VISUALIZATION VISU_Diagnostics  // 800x480
END_VISUALIZATION

(* stored: Version 1.1.0.1, ProductVersion 3.1.4026.18
   Visu VISU_Diagnostics: Id {38520286-8322-4592-931b-095319deec32} *)
